FUNCTION_BLOCK Motor
VAR_INPUT
END_VAR
VAR_OUTPUT
END_VAR
VAR
	interlock : BOOL;
	stop: BOOL;
	motor_select : INT := 0;
	mc1 : MotorControla;
	mc2 : MotorControla;
	mc3 : MotorControla;
	mc4 : MotorControla;
	tst: BOOL := FALSE;
	dmp: WORD;
END_VAR

//manual control
GVL.MDP := FALSE;
GVL.MIP := FALSE;
GVL.MPP := FALSE;
GVL.MVP := FALSE;
IF GVL.ToggleSwitch = TRUE THEN
	AUTO.Varno := FALSE;
	IF GVL.ULBButton THEN
		motor_select := 1;
	ELSIF GVL.URBButton THEN
		motor_select := 2;
	ELSIF GVL.LLBButton THEN
		motor_select := 3;
	ELSIF GVL.LRBButton THEN
		motor_select := 4;
	END_IF
	
	CASE motor_select OF
		1: mc1(
			Premik := GVL.RedButton,
			Smer := GVL.GreenButton,
			Select := TRUE,
			KS := GVL.KSV,
			Step :=GVL.StV,
			Limes := 185,
			Position => AUTO.Current.A,
			OutSmer => GVL.MVS,
			OutPremik => GVL.MVP,
			Interlock => interlock,
			Stop => stop
			);
		2: mc2(
			Premik := GVL.RedButton,
			Smer := GVL.GreenButton,
			Select := TRUE,
			KS := GVL.KSD,
			Step :=GVL.StD,
			Limes := 105,
			Position => AUTO.Current.Z,
			OutSmer => GVL.MDS,
			OutPremik => GVL.MDP,
			Interlock => interlock,
			Stop => stop);
		3: mc3(
			Premik := GVL.RedButton,
			Smer := GVL.GreenButton,
			Select := TRUE,
			KS := GVL.KSI,
			Step :=GVL.StI,
			Limes := 65,
			Position => AUTO.Current.Y,
			OutSmer => GVL.MIS,
			OutPremik => GVL.MIP,
			Interlock => interlock,
			Stop => stop);
		4: mc4(
			Premik := GVL.RedButton,
			Smer := GVL.GreenButton,
			Select := TRUE,
			KS := GVL.KSP,
			Step :=GVL.StP,
			Limes := 16,
			Position => AUTO.Current.P,
			OutSmer => GVL.MPS,
			OutPremik => GVL.MPP,
			Interlock => interlock,
			Stop => stop);
	END_CASE
	
	GVL.LEDGreen := stop;
	GVL.LEDRed := interlock;
	
ELSE
	CASE AUTO.MotorIzbira OF
		1: mc1(
			Premik := AUTO.VrtenjePremik,
			Smer := AUTO.VrtenjeSmer,
			Select := TRUE,
			KS := GVL.KSV,
			Step :=GVL.StV,
			Limes := 185,
			Position => AUTO.Current.A,
			OutPremik => GVL.MVP,
			OutSmer => GVL.MVS,
			Interlock => interlock,
			Stop => stop
			);
		2: mc2(
			Premik := AUTO.DvigPremik,
			Smer := AUTO.DvigSmer,
			Select := TRUE,
			KS := GVL.KSD,
			Step :=GVL.StD,
			Limes := 105,
			Position => AUTO.Current.Z,
			OutPremik => GVL.MDP,
			OutSmer => GVL.MDS,
			Interlock => interlock,
			Stop => stop
			);
		
		3: IF AUTO.Current.Y = 0 AND AUTO.IztegSmer = TRUE THEN
			//GVL.LEDLBlue := TRUE;
			ELSE
			//.LEDLBlue := FALSE;
			mc3(
			Premik := AUTO.IztegPremik,
			Smer := AUTO.IztegSmer,
			Select := TRUE,
			KS := GVL.KSI,
			Step :=GVL.StI,
			Limes := 60,
			Position => AUTO.Current.Y,
			OutPremik => GVL.MIP,
			OutSmer => GVL.MIS,
			Interlock => interlock,
			Stop => stop
			);
			END_IF
		4: mc4(
			Premik := AUTO.PrijemPremik,
			Smer := AUTO.PrijemSmer,
			Select := TRUE,
			KS := GVL.KSP,
			Step :=GVL.StP,
			Limes := 16,
			Position => AUTO.Current.P,
			OutPremik => GVL.MPP,
			OutSmer => GVL.MPS,
			Interlock => interlock,
			Stop => stop
			);
	END_CASE
	
	GVL.LEDGreen := stop;
	GVL.LEDRed := interlock;
	
END_IF

RETURN;

END_FUNCTION_BLOCK

(* stored: Version 1.1.0.1, ProductVersion 3.1.4024.12
   POU Motor: Id {183a81e9-a3e5-4857-ba31-4a4bf27437fb}, SpecialFunc None *)
